INTERFACE I_RpcParameters

METHOD PUBLIC TryCopyStringParameter : BOOL;
VAR_INPUT
	ParameterName : STRING;
	DestinationAddress : REFERENCE TO STRING;
	DestinationSize : UDINT;
END_VAR
END_METHOD

METHOD PUBLIC TryGetParameter : BOOL;
VAR_INPUT
	ParameterName : STRING;
	Destination : ANY;
END_VAR
END_METHOD

METHOD PUBLIC TryGetStringParameterSize : BOOL;
VAR_INPUT
	ParameterName : STRING;
	Destination : REFERENCE TO UDINT;	
END_VAR
END_METHOD

END_INTERFACE

(* stored: Version 1.1.0.1, ProductVersion 3.1.4024.12
   Itf I_RpcParameters: Id {d229831f-509a-4603-8f9f-3929e2ad8d48}
   Method TryCopyStringParameter: Id {c1a81c98-cb01-414b-9bca-d02d8cd54dcc}
   Method TryGetParameter: Id {3a562980-8096-4409-9c13-3d2c6a091a24}
   Method TryGetStringParameterSize: Id {e31772a3-49da-41c1-8e1b-af7cb802bafa} *)
